(* Schneider Machine Expert - Basic project Conveyors, file version 2.2.0.0 *)
(* ProjectInformations: Name=New project *)

HARDWARE
  Cpu 0: TM221M16R/G
  EthernetConfiguration: NetworkName=M221, IpAllocationMode=FixedAddress, IpAddress=0.0.0.0, SubnetMask=0.0.0.0
  SerialLineConfiguration: Baud=Baud19200, Parity=ParityEven, DataBits=DataBits8, StopBits=StopBits1, PhysicalMedium=PhysicalMediumRs485, TransmissionMode=TransmissionModeModbusRtu, SlaveId=1, Addressing=SlaveAddressing
  MastTask: UsePeriodScanMode=false, PeriodScan=100
  FastTask: Period=255
  CpuBehavior: StartingMode=StartAsPreviousState, AutoSaveRamOnEeprom=true, WatchdogPeriod=250

SYMBOLS  (address, symbol, comment, settings)
  %M100     RUN_RE
  %M105     C1_FLTR
  %M106     C2_FLTR
  %M107     C3_FLTR
  %M109     STOP_R
  %S6       SB_TB1S  "Time base of 1 s generated by an internal clock"
  %I0.6     STOP_BUTTON
  %I0.7     START_BUTTON
  %Q0.2     C1_RUN
  %Q0.4     C3_RUN
  %Q0.6     RUN_LIGHT

POU Control
  (* SectionNumber=1 *)

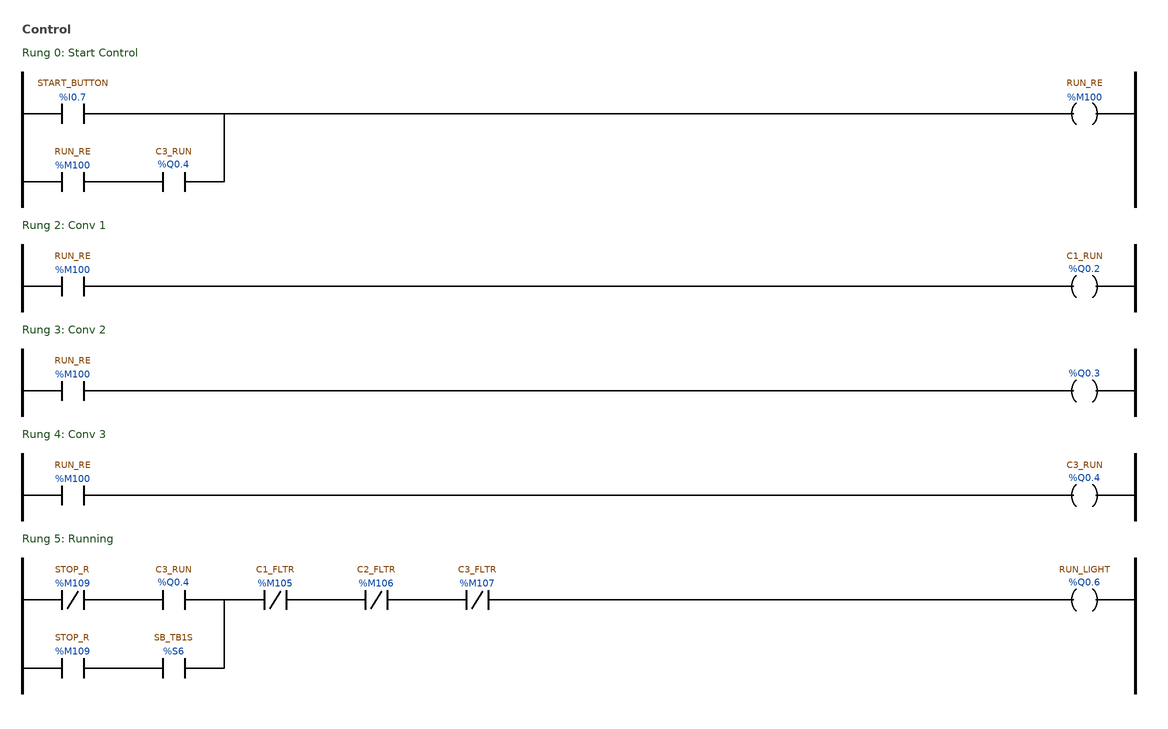

// Rung 0: Start Control
  LD %I0.7                (* START_BUTTON *)
  OR( %M100               (* RUN_RE *)
  AND %Q0.4               (* C3_RUN *)
  )
  ST %M100                (* RUN_RE *)
  // as ST:
  //   RUN_RE := START_BUTTON OR RUN_RE AND C3_RUN;

// Rung 1: Stop Control
  LD

// Rung 2: Conv 1
  LD %M100                (* RUN_RE *)
  ST %Q0.2                (* C1_RUN *)
  // as ST:
  //   C1_RUN := RUN_RE;

// Rung 3: Conv 2
  LD %M100                (* RUN_RE *)
  ST %Q0.3
  // as ST:
  //   %Q0.3 := RUN_RE;

// Rung 4: Conv 3
  LD %M100                (* RUN_RE *)
  ST %Q0.4                (* C3_RUN *)
  // as ST:
  //   C3_RUN := RUN_RE;

// Rung 5: Running
  LDN %M109               (* STOP_R *)
  AND %Q0.4               (* C3_RUN *)
  OR( %M109               (* STOP_R *)
  AND %S6                 (* SB_TB1S *)
  )
  ANDN %M105              (* C1_FLTR *)
  ANDN %M106              (* C2_FLTR *)
  ANDN %M107              (* C3_FLTR *)
  ST %Q0.6                (* RUN_LIGHT *)
  // as ST:
  //   RUN_LIGHT := (NOT STOP_R AND C3_RUN OR STOP_R AND SB_TB1S) AND NOT C1_FLTR AND NOT C2_FLTR AND NOT C3_FLTR;

// Rung 6: Stop 1
  LD

// Rung 7: Stop 2
  LD

// Rung 8: Stop 3
  (* no IL stored for this rung *)

POU Speed Monitoring
  (* SectionNumber=2 *)

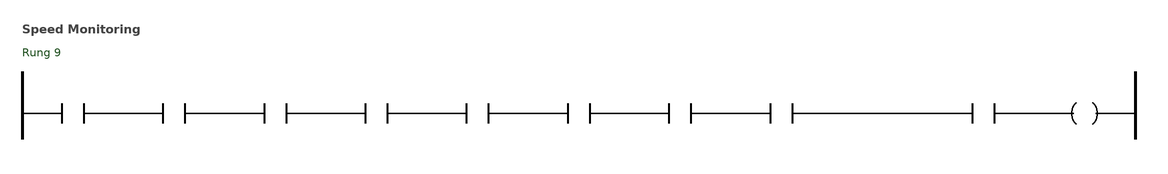

// Rung 9
  (* no IL stored for this rung *)

POU Fault Handling
  (* SectionNumber=3 *)

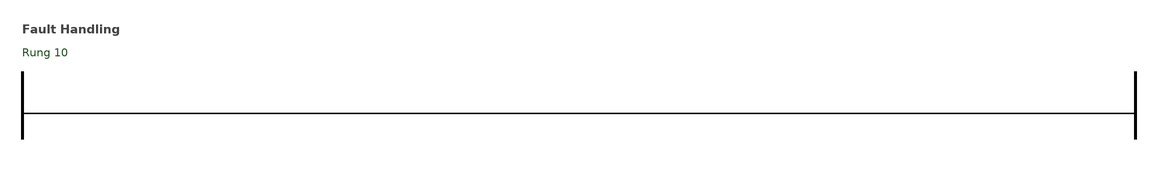

// Rung 10
  (* no IL stored for this rung *)
